RoboDK station: Stringer B-Top2-BOX2.rdk

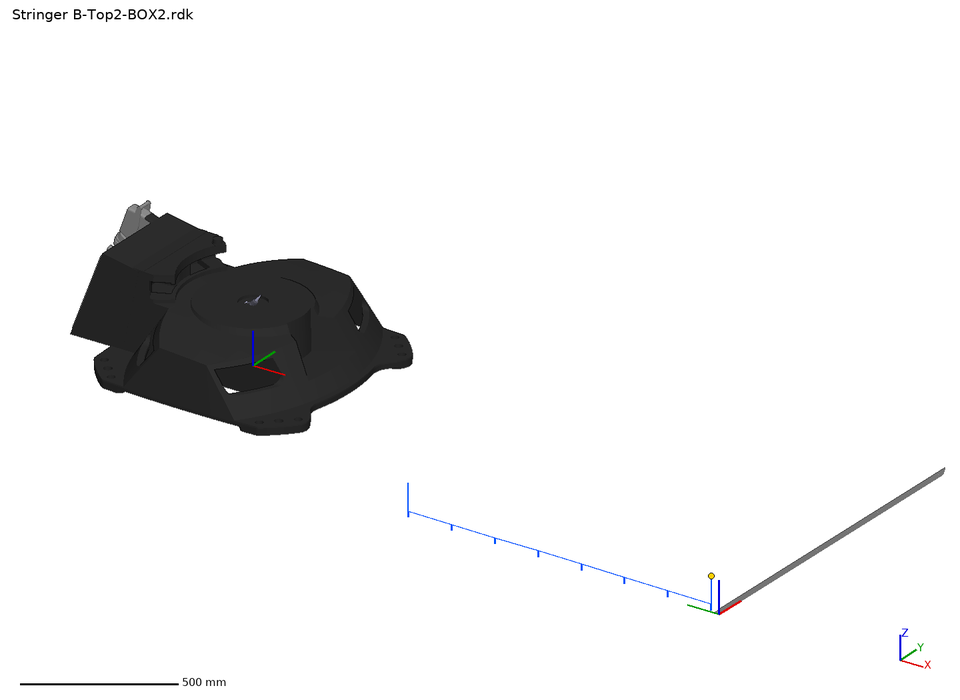
[picture v0: the station drawn from its stored meshes, robots at their saved joint values, targets as dots, program paths as lines]
Station Stringer B-Top2-BOX2 (saved by RoboDK 5.2.3). Poses are relative to the parent item; angles as X-Y-Z fixed-axis rotations.
  - frame KUKA KR 210 R2700 extra Base at (0, 0, 0) mm
    - robot KUKA KR 210 R2700 extra: 6 axes, payload 210 kg, reach 2696 mm, repeatability 0.06 mm, weight 1068 kg
        joint limits [-185, -140, -120, -350, -125, -350] to [185, -5, 155, 350, 125, 350]; home [0, -90, 90, 0, 0, 0]; saved at [-38.593, -26.987, 87.041, 95.566, 23.23, -127.863]
      - tool Spindle, TCP at (32, 0, 260) mm, rotated rx 0 ry 39 rz 0 deg, size 157.3 x 72 x 259.9 mm
  - frame Frame 2 at (1800, 0, -372.68) mm, rotated rx 0 ry 0 rz 90 deg
    - object Stringer B-Top2-BOX2 at (0, 22.5, 0) mm, rotated rx 0 ry 0 rz -90 deg, 8 curves, geometry from Point 8
    - object L-Stringer B -Top2-BOX2 at (0, 0, 0) mm, size 1245.4 x 20 x 20 mm, geometry from L-Stringer B -Top2-BOX2.stl
  - machining project Point settings: rotZ(0) | rotX(0)*rotY(0) | rotz(0) | onStart | onPathStart | onApproach | onPoint | onRetract | onFinish | SetRPM(%1) | SetTool(%1) | Extruder(%1) | default | default | OutOnMov(%1) | OutOffMov(%1) | onPathFinish | M_RunCode(%1)
  - program Point (51 instructions, listed below)
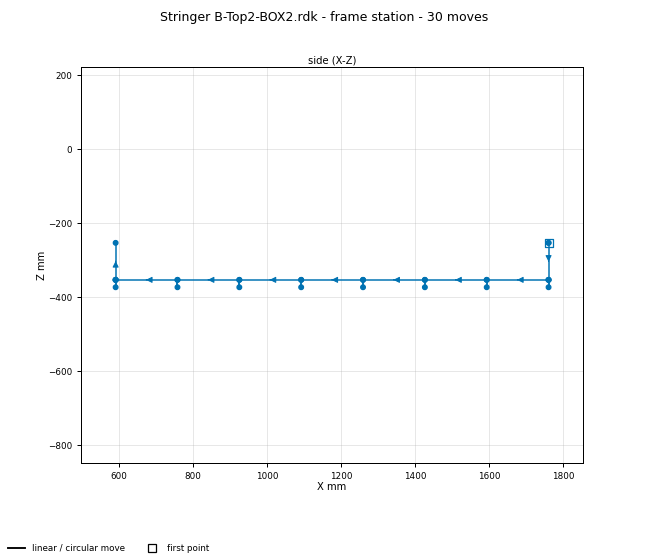
[picture p0: tool path of Stringer B-Top2-BOX2.rdk in frame station, 30 of 30 moves have a stored position in this frame; points joined in program order, loops and branches not executed]

--- program Point (robot KUKA KR 210 R2700 extra) ---
  Smooth(1)
  Set speed (1000.0 mm/s)
  Set Ref.: Frame 2
  Set Tool: Spindle
  Show Spindle
  MoveJ 1 to (11.5, 39.08, 120) mm, rotated rx -180 ry 0 rz -180 deg; joints [-1.478, -34.019, 111.88, 177.942, 26.866, -179.312]
  MoveL 2 to (11.5, 39.08, 120) mm, rotated rx -180 ry 0 rz -180 deg; joints [-1.478, -34.019, 111.88, 177.942, 26.866, -179.312]
  MoveL 3 to (11.5, 39.08, 20) mm, rotated rx 180 ry 0 rz 180 deg; joints [-1.478, -28.688, 109.236, 178.114, 29.553, -179.508]
  MoveL 4 to (11.5, 39.08, 20) mm, rotated rx 180 ry 0 rz 180 deg; joints [-1.478, -28.688, 109.236, 178.114, 29.553, -179.508]
  Set speed (50.0 mm/s)
  MoveL 5 to (11.5, 39.08, 0) mm, rotated rx -180 ry 0 rz -180 deg; joints [-1.478, -27.63, 108.66, 178.142, 30.034, -179.54]
  MoveL 6 to (11.5, 39.08, 20) mm, rotated rx 180 ry 0 rz 180 deg; joints [-1.478, -28.688, 109.236, 178.114, 29.553, -179.508]
  Set speed (1000.0 mm/s)
  MoveL 7 to (11.5, 206.23, 20) mm, rotated rx 180 ry 0 rz 180 deg; joints [-7.752, -28.59, 108.535, 169.936, 29.064, -177.221]
  Set speed (50.0 mm/s)
  MoveL 8 to (11.5, 206.23, 0) mm, rotated rx 180 ry 0 rz 180 deg; joints [-7.752, -27.539, 107.962, 170.084, 29.535, -177.391]
  MoveL 9 to (11.5, 206.23, 20) mm, rotated rx 180 ry 0 rz 180 deg; joints [-7.752, -28.59, 108.535, 169.936, 29.064, -177.221]
  Set speed (1000.0 mm/s)
  MoveL 10 to (11.5, 373.37, 20) mm, rotated rx -180 ry 0 rz -180 deg; joints [-13.845, -28.337, 106.885, 161.287, 27.994, -174.19]
  Set speed (50.0 mm/s)
  MoveL 11 to (11.5, 373.37, 0) mm, rotated rx 180 ry 0 rz 180 deg; joints [-13.845, -27.299, 106.317, 161.565, 28.44, -174.507]
  MoveL 12 to (11.5, 373.37, 20) mm, rotated rx -180 ry 0 rz -180 deg; joints [-13.845, -28.337, 106.885, 161.287, 27.994, -174.19]
  Set speed (1000.0 mm/s)
  MoveL 13 to (11.5, 540.51, 20) mm, rotated rx -180 ry 0 rz -180 deg; joints [-19.636, -27.875, 104.295, 151.756, 26.544, -169.83]
  Set speed (50.0 mm/s)
  MoveL 14 to (11.5, 540.51, 0) mm, rotated rx 180 ry 0 rz 180 deg; joints [-19.636, -26.859, 103.735, 152.182, 26.946, -170.307]
  MoveL 15 to (11.5, 540.51, 20) mm, rotated rx -180 ry 0 rz -180 deg; joints [-19.636, -27.875, 104.295, 151.756, 26.544, -169.83]
  Set speed (1000.0 mm/s)
  MoveL 16 to (11.5, 707.66, 20) mm, rotated rx 180 ry 0 rz -180 deg; joints [-25.038, -27.138, 100.778, 140.938, 25.003, -163.617]
  Set speed (50.0 mm/s)
  MoveL 17 to (11.5, 707.66, 0) mm, rotated rx -180 ry 0 rz -180 deg; joints [-25.038, -26.149, 100.227, 141.522, 25.345, -164.262]
  MoveL 18 to (11.5, 707.66, 20) mm, rotated rx 180 ry 0 rz -180 deg; joints [-25.038, -27.138, 100.778, 140.938, 25.003, -163.617]
  Set speed (1000.0 mm/s)
  MoveL 19 to (11.5, 874.8, 20) mm, rotated rx -180 ry 0 rz -180 deg; joints [-30.004, -26.053, 96.337, 128.56, 23.731, -155.217]
  Set speed (50.0 mm/s)
  MoveL 20 to (11.5, 874.8, 0) mm, rotated rx 180 ry 0 rz -180 deg; joints [-30.004, -25.094, 95.794, 129.291, 23.993, -156.017]
  MoveL 21 to (11.5, 874.8, 20) mm, rotated rx -180 ry 0 rz -180 deg; joints [-30.004, -26.053, 96.337, 128.56, 23.731, -155.217]
  Set speed (1000.0 mm/s)
  MoveL 22 to (11.5, 1041.94, 20) mm, rotated rx -180 ry 0 rz -180 deg; joints [-34.519, -24.547, 90.96, 114.726, 23.118, -144.722]
  Set speed (50.0 mm/s)
  MoveL 23 to (11.5, 1041.94, 0) mm, rotated rx 180 ry 0 rz 180 deg; joints [-34.519, -23.618, 90.421, 115.55, 23.283, -145.618]
  MoveL 24 to (11.5, 1041.94, 20) mm, rotated rx -180 ry 0 rz -180 deg; joints [-34.519, -24.547, 90.96, 114.726, 23.118, -144.722]
  Set speed (1000.0 mm/s)
  MoveL 25 to (11.5, 1209.08, 20) mm, rotated rx -180 ry 0 rz -180 deg; joints [-38.593, -22.543, 84.597, 100.155, 23.504, -132.861]
  Set speed (50.0 mm/s)
  MoveL 26 to (11.5, 1209.08, 0) mm, rotated rx 180 ry 0 rz 180 deg; joints [-38.593, -21.644, 84.058, 100.967, 23.57, -133.746]
  MoveL 27 to (11.5, 1209.08, 20) mm, rotated rx -180 ry 0 rz -180 deg; joints [-38.593, -22.543, 84.597, 100.155, 23.504, -132.861]
  MoveL 28 to (11.5, 1209.08, 20) mm, rotated rx -180 ry 0 rz -180 deg; joints [-38.593, -22.543, 84.597, 100.155, 23.504, -132.861]
  Set speed (1000.0 mm/s)
  MoveL 29 to (11.5, 1209.08, 20) mm, rotated rx -180 ry 0 rz -180 deg; joints [-38.593, -22.543, 84.597, 100.155, 23.504, -132.861]
  MoveL 30 to (11.5, 1209.08, 120) mm, rotated rx -180 ry 0 rz -180 deg; joints [-38.593, -26.987, 87.041, 95.566, 23.23, -127.863]
